Universal Robots PolyScope program: Robot1.urp

Program Robot1 (installation=default directory=/programs/usbdisk_0 createdIn=5.12.0.1101482 lastSavedIn=5.12.0.1101482 robotSerialNumber=20215600259)
Calibrated DH parameters: a=[0.000144, -0.229031, -0.356292, 0.000082, -0.000021, 0]; d=[0.180658, -276.462654, 291.096579, -14.459979, 0.119851, 0.115626]; alpha=[1.571461, 0.001518, -0.00357, 1.569954, -1.570852, 0]; deltaTheta=[0, -1.071167, 7.208741, 0.145613, 0, 0]
Robot Program (runOnlyOnce=false)
  MoveL speed 150 mm/s, acceleration 2 mm/s^2 (useActiveTCP=true) feature=Base
    Waypoint Контр_точка_1: motionParameters(jointSpeed=1.047198 jointAcceleration=1.396263 cartesianSpeed=0.8 cartesianAcceleration=0.1); TCP in base x=159.193 y=-442.906 z=694.444 mm, rx=-0.0242 ry=-3.1406 rz=-0.0075 rad; joints [88.099, -84.269, 43.132, -48.592, -90.227, -0.864] deg; TCP offset x=0 y=0 z=83 mm, rx=0 ry=0 rz=0 rad
    Waypoint Контр_точка_2: motionParameters(jointSpeed=1.047198 jointAcceleration=1.396263 cartesianSpeed=0.8 cartesianAcceleration=0.1); TCP in base x=148.177 y=-770.704 z=-212.484 mm, rx=0.1313 ry=-3.134 rz=0.0046 rad; joints [88.23, -14.078, 73.909, -150.023, -90.329, -6.763] deg
    MoveDirectionNode (selectedDirection=ZPlus toolParams=0.5, 0.0065) feature=Joint_6_name
      Until TOOL_CONTACT_DETECTION (allowActions=false retraction=0.002 decelerationAcceleration=0.3 decelerationAngularAcceleration=34.906585)
    URCap VG Захват (OnRobot, OnRobot A/S) dataModel(vg.channel.a=true, vg.grip.req.channel.a=true, vg.channel.b=true, vg.grip.req.channel.b=true, vg.grip.seek=true, Variable(key=on_return, variable(name=on_return)))
    MoveDirectionNode (selectedDirection=ZMinus toolParams=0.8, 0.1) feature=Joint_6_name
      Until DISTANCE (allowActions=false deceleration=3 distanceNodeType=STOP) Distance=0.12; motionParameters(blendRadius=0)
    MoveDirectionNode (toolParams=1.2, 0.1) expression=[75.0,100.0,0.0]; feature=Base
      Until DISTANCE (allowActions=false deceleration=3 distanceNodeType=STOP) Distance=1; motionParameters(blendRadius=0.25)
    MoveDirectionNode (selectedDirection=ZPlus toolParams=0.3, 0.01) feature=Joint_6_name
      Until TOOL_CONTACT_DETECTION (allowActions=false retraction=0.007 decelerationAcceleration=0.225 decelerationAngularAcceleration=34.906585)
    URCap VG Отпускание (OnRobot, OnRobot A/S)
  MoveP speed 250 mm/s, acceleration 1200 mm/s^2 (blendRadius=0.025 useActiveTCP=true) feature=Base
    MoveDirectionNode (selectedDirection=ZMinus toolParams=0.8, 0.1) feature=Joint_6_name
      Until DISTANCE (allowActions=false deceleration=3 distanceNodeType=STOP) Distance=0.3; motionParameters(blendRadius=0)
